{attribute 'qualified_only'}
{attribute 'strict'}
TYPE E_PISTON_TYPE :
(
	NO_SENSORS,
	ONLY_OPEN,
	ONLY_CLOSE,
	BOTH
);
END_TYPE

(* stored: Version 1.1.0.1, ProductVersion 3.1.4024.12
   DUT E_PISTON_TYPE: Id {609b13fd-83ea-4c41-a20b-05c2b0faa5b2} *)
